{attribute 'qualified_only'}
{attribute 'strict'}
TYPE E_LED_MODES :
(
	// SOLID ODD; FLASH EVEN
	OFF := -1,
    YELLOW := 1,
    RED := 2,
	GREEN := 3
);
END_TYPE

(* stored: Version 1.1.0.1, ProductVersion 3.1.4024.12
   DUT E_LED_MODES: Id {86f86d08-88f0-44ab-bd2a-e10eac74146c} *)
